FUNCTION_BLOCK SYS_ONTIME (* Service Interface Function Block Type *)
  (* Standard: 61499-2; Description: Copyright (c) 2025 HR Agrartechnik GmbH This program and the accompanying materials are made available under the terms of the Eclipse Public License 2.0 which is available at https://www.eclipse.org/legal/epl-2.0/ SPDX-License-Identifier: EPL-2.0 *)
  (* Version 1.0, 2025-05-02, Franz Höpfinger, HR Agrartechnik GmbH, initial API and implementation and/or initial documentation *)
  PACKAGE logiBUS::signalprocessing::measurement;
  IMPORT eclipse4diac::core::TypeHash;
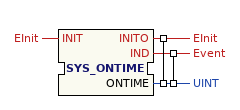
  EVENT_INPUT
    INIT : EInit; (* Service Initialization *)
  END_EVENT
  EVENT_OUTPUT
    INITO : EInit WITH ONTIME; (* Initialization Confirm *)
    IND WITH ONTIME; (* Indication from Resource *)
  END_EVENT
  VAR_OUTPUT
    ONTIME : UINT; (* Input data from resource: ONTIME in Decimal minute (0.01 Hours) *)
  END_VAR
END_FUNCTION_BLOCK
